TYPE ST_INPUTS_Unit_UltraSonCleaner:
STRUCT
	
	Mode:     		E_DeviceMode;
	Command:     E_DeviceState;

END_STRUCT
END_TYPE

(* stored: Version 1.1.0.1, ProductVersion 3.1.4024.12
   DUT ST_INPUTS_Unit_UltraSonCleaner: Id {39599569-8f20-491b-b695-42a364e749dc} *)
